SUBAPPLICATION mapping_Uebung_003c (* DigitalInput_I1-2-3-4 auf AUX *)
  (* Standard: 61499-2; Description: Copyright (c) 2023 Meisterschulen am Ostbahnhof This program and the accompanying materials are made available under the terms of the Eclipse Public License 2.0 which is available at https://www.eclipse.org/legal/epl-2.0/ SPDX-License-Identifier: EPL-2.0 *)
  (* Version 1.0, 2023-10-23, Franz Höpfinger, Meisterschulen am Ostbahnhof *)
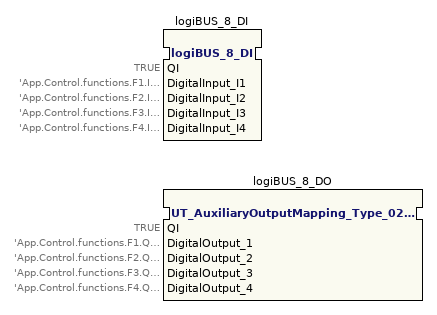
  FBS
    logiBUS_8_DO : UT_AuxiliaryOutputMapping_Type_02_Bool_NonLatched(QI := TRUE, DigitalOutput_1 := 'App.Control.functions.F1.QX', DigitalOutput_2 := 'App.Control.functions.F2.QX', DigitalOutput_3 := 'App.Control.functions.F3.QX', DigitalOutput_4 := 'App.Control.functions.F4.QX');
    logiBUS_8_DI : logiBUS_8_DI(QI := TRUE, DigitalInput_I1 := 'App.Control.functions.F1.IX', DigitalInput_I2 := 'App.Control.functions.F2.IX', DigitalInput_I3 := 'App.Control.functions.F3.IX', DigitalInput_I4 := 'App.Control.functions.F4.IX');
  END_FBS
END_SUBAPPLICATION
